{attribute 'qualified_only'}
{attribute 'strict'}
TYPE E_FqInverterState :
(
	DISABLED,
	ENABLED,
	RUNNING,
	ERROR,
	RESET
);
END_TYPE

(* stored: Version 1.1.0.1, ProductVersion 3.1.4024.14
   DUT E_FqInverterState: Id {f05ed465-757d-070d-1b89-908f7a1a7525} *)
